FUNCTION_BLOCK For
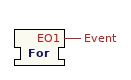
  EVENT_OUTPUT
    EO1;
  END_EVENT
  EC_STATES
    START;
    S2 : A1 -> EO1;
  END_STATES
  ALGORITHM A1 IN ST:
  VAR_TEMP
    sum : INT;
    i : INT;
  END_VAR
FOR i := 0 TO 10 DO&#38;#10;  sum := sum + i;&#38;#10;END_FOR;&#38;#10;
  END_ALGORITHM
END_FUNCTION_BLOCK
